//==============================Get Ready after actio finished ===========
      A     #sqSequencer.STEP.ActionFinished;
      JCN   k011;
// Reset Action finished flag, ready for next step action
      R     #sqSequencer.STEP.ActionVerified;
      R     #sqSequencer.STEP.ActionFinished;
//======================if ALL actions are finished========================
      SET   ;
      S     #sqSequencer.STEP.Finished;
      R     #sqSequencer.STEP.Active;
      S     #sqSequencer.STEP.Done[11];
//=====================End Step action(s)==================================
      JU    k011;
//===========================Finished Step Action(s)======================
k011: NOP   0;

      A     #sqStepTimer.Q;
      S     #sqSequencer.STEP.WithError[11]; // Step error flag
      S     #sqSequencer.Error_Fault;
      R     #sqStepTimer.IN;
NETWORK
TITLE =S011:STEP-011::Begin Transition

A011: NOP   0;
     R     #sqStepTimer.IN;






NETWORK
TITLE =S011::STEP-011:EXIT TRANSITION:
//--------------------------------------------------------------------------
// Jump to the common step progression code:
//--------------------------------------------------------------------------
      JU    COMM;







NETWORK
TITLE =Sequencer Common Code, Execute in Each Scan

COMM: NOP   0;


NETWORK
TITLE =Retentive/Non Retentive Selectable Run timer

      CALL #sqRunTimer (
           TIME_H                   := #sqRunTimer.TIME_H,
           TIME_M                   := #sqRunTimer.TIME_M,
           TIME_S                   := #sqRunTimer.TIME_S,
           ENABLE                   := #sqRunTimer.ENABLE,
           RESET                    := #sqRunTimer.RESET,
           PAUSE                    := #sqRunTimer.PAUSE,
           NON_RET                  := #sqRunTimer.NON_RET,
           RMNG_H                   := #sqRunTimer.RMNG_H,
           RMNG_M                   := #sqRunTimer.RMNG_M,
           RMNG_S                   := #sqRunTimer.RMNG_S,
           TIME_EXPIRED             := #sqRunTimer.TIME_EXPIRED,
           TMR_RUNNG                := #sqRunTimer.TMR_RUNNG);


NETWORK
TITLE =Sequencer Step Timer

      CALL #sqStepTimer (
           IN                       := #sqStepTimer.IN,
           PT                       := "dbCONST_VAL".SQ_STEP_TIME,
           Q                        := #sqStepTimer.Q,
           ET                       := #sqStepTimer.ET);


NETWORK
TITLE =Sequencer Timer

 CALL #SQ_TIMER (
           IN                       := #SQ_TIMER.IN,
           PT                       := #SQ_TIMER.PT,
           Q                        := #SQ_TIMER.Q,
           ET                       := #SQ_TIMER.ET);


NETWORK
TITLE =General Assignments

      L     #sqSequencer.STEP.NumberNext;
      T     #NXT_STEP;
      T     #sqSequencer.STEP.NumberCurrent;
      T     #CURSTEP;


      A     #sqSequencer.STEP.Active;
      =     #S_ACTIVE;


      A     #sqSequencer.Error_Fault;
      =     #ERR_FAULT;

NETWORK
TITLE =Sequencer Finished


      AN    #OFF_IDLE;
      AN    #PAUSED;
      A     #sqSequencer.STEP.Done[11];
      =     #sqSequencer.Finished;
      =     #SQ_FINISHED;
      JCN   fnsd;
      L     "dbCONST_VAL".SQ_STATE.COMPLETE;
      T     #SQ_STATE;
      R     #PAUSED;
      R     #sqSequencer.STEP.Error_Fault;
      R     #sqSequencer.Error_Fault;
fnsd: NOP   0;


//Reset Finished flag if SQ OFF for Last step to scan.
      A     #OFF_IDLE;
      AN    #sqSequencer.STEP.Done[11];
      AN    #sqSequencer.STEP.WithError[11];
      JCN   abrt;
      R     #sqSequencer.STEP.Finished;
      L     "dbCONST_VAL".SQ_STATE.ABORTED;
      T     #SQ_STATE;
      S     #OFF_IDLE;
      R     #PAUSED;
      R     #sqSequencer.STEP.Error_Fault;
      R     #sqSequencer.Error_Fault;
      R     #PAUSED;
abrt: NOP   0;





//========================Visio Common Code Begin===========================


//========================Visio Common Code End===========================
//End of Sequencer





END_FUNCTION_BLOCK


